FUNCTION_BLOCK XtsTrack IMPLEMENTS IXtsTrack
VAR_INPUT
	StateMachine : IPmlStateMachine;
END_VAR
VAR_OUTPUT
END_VAR
VAR
	_trackLength : MC_LREAL := 8000.0;
	mcCollisionGroup : CollisionGroup;
	XtsTrackHardware : XtsHardware;
	EnableSequence : XtsEnableSequence(mcCollisionGroup);
	DisableSequence : XtsDisableSequence(mcCollisionGroup);
	State :(
        Init,                                               
		Ready,                                 
        Enabling,
		Enabled,
		Resetting,
		Running,
		Disabling);  	
	i : DINT;
	AtHome: BOOL;
END_VAR
VAR_IN_OUT
	MoverArray : ARRAY[*] OF IMover;
END_VAR

XtsTrackHardware();
CASE State OF
	Init:
		IF XtsTrackHardware.XtsHardwareOK THEN
			State := Ready;
		END_IF
		
	Ready:
		IF StateMachine.getState() = E_PMLState.ePMLState_Clearing THEN
			IF EnableSequence.Enable() THEN
				State := Enabling;
			END_IF	
		END_IF
		
	Enabling:
		IF EnableSequence.Done THEN
			State := Enabled;
			StateMachine.StateComplete();
		END_IF
		
	Enabled:
		IF StateMachine.getState() = E_PMLState.ePMLState_Aborting THEN
			DisableSequence.Disable();
			IF DisableSequence.Busy THEN
				State := Disabling;
			END_IF
		END_IF
		
		IF StateMachine.getState() = E_PMLState.ePMLState_Resetting THEN
			FOR i := LOWER_BOUND(MoverArray,1) TO UPPER_BOUND(MoverArray,1) DO
				MoverArray[i].MoveTo(Position := 5500.0, Velocity := 1000.0, BackwardMove := FALSE);
			END_FOR 
			State := Resetting;
		END_IF
		
	Resetting:
		AtHome := TRUE;
		FOR i := LOWER_BOUND(MoverArray,1) TO UPPER_BOUND(MoverArray,1) DO
				AtHome := AtHome AND MoverArray[i].isStationary();
		END_FOR 
		IF AtHome THEN
			State := Running;
			StateMachine.StateComplete();	
		END_IF
		
	Running:	
		IF StateMachine.getState() = E_PMLState.ePMLState_Aborting THEN
			DisableSequence.Disable();
			IF DisableSequence.Busy THEN
				State := Disabling;
			END_IF
		END_IF
		
	Disabling:
		IF DisableSequence.Done THEN
			State := Ready;
			StateMachine.StateComplete();
		END_IF
	
END_CASE

EnableSequence(arrMovers := MoverArray);
DisableSequence(arrMovers := MoverArray);
mcCollisionGroup();

PROPERTY PUBLIC TrackLength : mc_lreal
GET
TrackLength := _trackLength;
END_GET
END_PROPERTY

END_FUNCTION_BLOCK

(* stored: Version 1.1.0.1, ProductVersion 3.1.4024.9
   POU XtsTrack: Id {cc8fa43e-3905-4147-a69e-0a5caa88babb}, SpecialFunc None
   Property TrackLength: Id {650984a1-6668-4032-bccb-d14c7a46cb5a}
   Get Get: Id {074949c2-3a12-4fc2-a08c-82a02f06bf44} *)
